TYPE ST_CYLINDER_Control :
STRUCT
	eCommand		: E_CYLINDER_Position;
END_STRUCT
END_TYPE

(* stored: Version 1.1.0.1, ProductVersion 3.1.4024.15
   DUT ST_CYLINDER_Control: Id {9cdf542e-e54b-4762-8636-a0df942675c3} *)
